// TODO rename + your recipe members. SchemaVersion is MANDATORY (Core §3.8).
TYPE ST_TemplateParCfg :
STRUCT
    SchemaVersion : UINT := 1;
    MoveTimeout   : TIME := T#2S;
END_STRUCT
END_TYPE

(* stored: Version 1.1.0.1, ProductVersion 3.1.4024.12
   DUT ST_TemplateParCfg: Id {d35ee904-798e-40d7-9c16-c050f4ec2ef5} *)
